(* PLC project One Station VGP, Blank VGP 1.0 *)
(* stored: creationDateTime 2016-05-18T21:14:07, modificationDateTime 2020-03-26T18:29:31 *)

FUNCTION ConvertPressure : SINT
  VAR_INPUT
    Pressure_input : UINT;
  END_VAR
  VAR_OUTPUT
    Pressure_output : INT;
  END_VAR
  VAR
    Pressure_real : LREAL;
  END_VAR

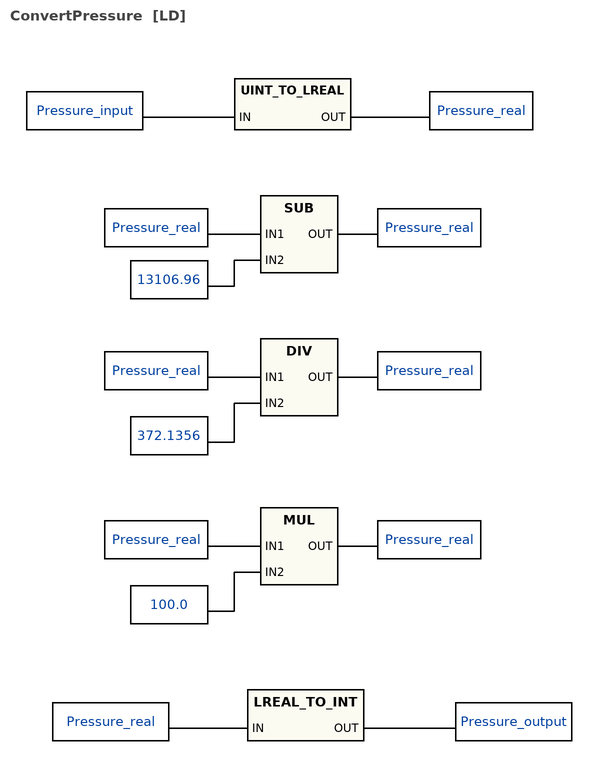
(* LD diagram, written out as Structured Text *)
Pressure_real := UINT_TO_LREAL(Pressure_input);
Pressure_real := Pressure_real - 13106.96;
Pressure_real := Pressure_real / 372.1356;
Pressure_real := Pressure_real * 100.0;
Pressure_output := LREAL_TO_INT(Pressure_real);
END_FUNCTION

PROGRAM My_Program
  VAR
    pressure AT %IW0 : UINT;
    pressure_psi AT %QW6 : INT;
    min_sp AT %QW1 : INT;
    max_sp AT %QW2 : INT;
  END_VAR
  VAR
    pump_mode : BOOL;
    pm_pump : BOOL;
    pm_valve : BOOL;
    valve_mode : BOOL;
    vm_pump : BOOL;
    vm_valve : BOOL;
    manual_mode : BOOL;
    mm_pump : BOOL;
    mm_valve : BOOL;
  END_VAR
  VAR
    mode_register AT %QW3 : INT;
    pump_register AT %QW4 : INT;
    valve_register AT %QW5 : INT;
  END_VAR
  VAR
    over_pressure : BOOL;
  END_VAR
  VAR
    pump AT %QX0.0 : BOOL;
    valve AT %QX0.1 : BOOL;
  END_VAR
  VAR
    TOF0 : TOF;
  END_VAR
  VAR  (* added by the conversion: wires and edge detectors of the diagram *)
    _LE4_ENO : BOOL;
    _LE4_OUT : BOOL;
    _GE11_ENO : BOOL;
    _GE11_OUT : BOOL;
    _LE22_ENO : BOOL;
    _LE22_OUT : BOOL;
    _GE29_ENO : BOOL;
    _GE29_OUT : BOOL;
    _EQ44_ENO : BOOL;
    _EQ44_OUT : BOOL;
    _EQ50_ENO : BOOL;
    _EQ50_OUT : BOOL;
    _ConvertPressure99_Pressure_output : ANY;
    _ConvertPressure99_OUT : SINT;
  END_VAR

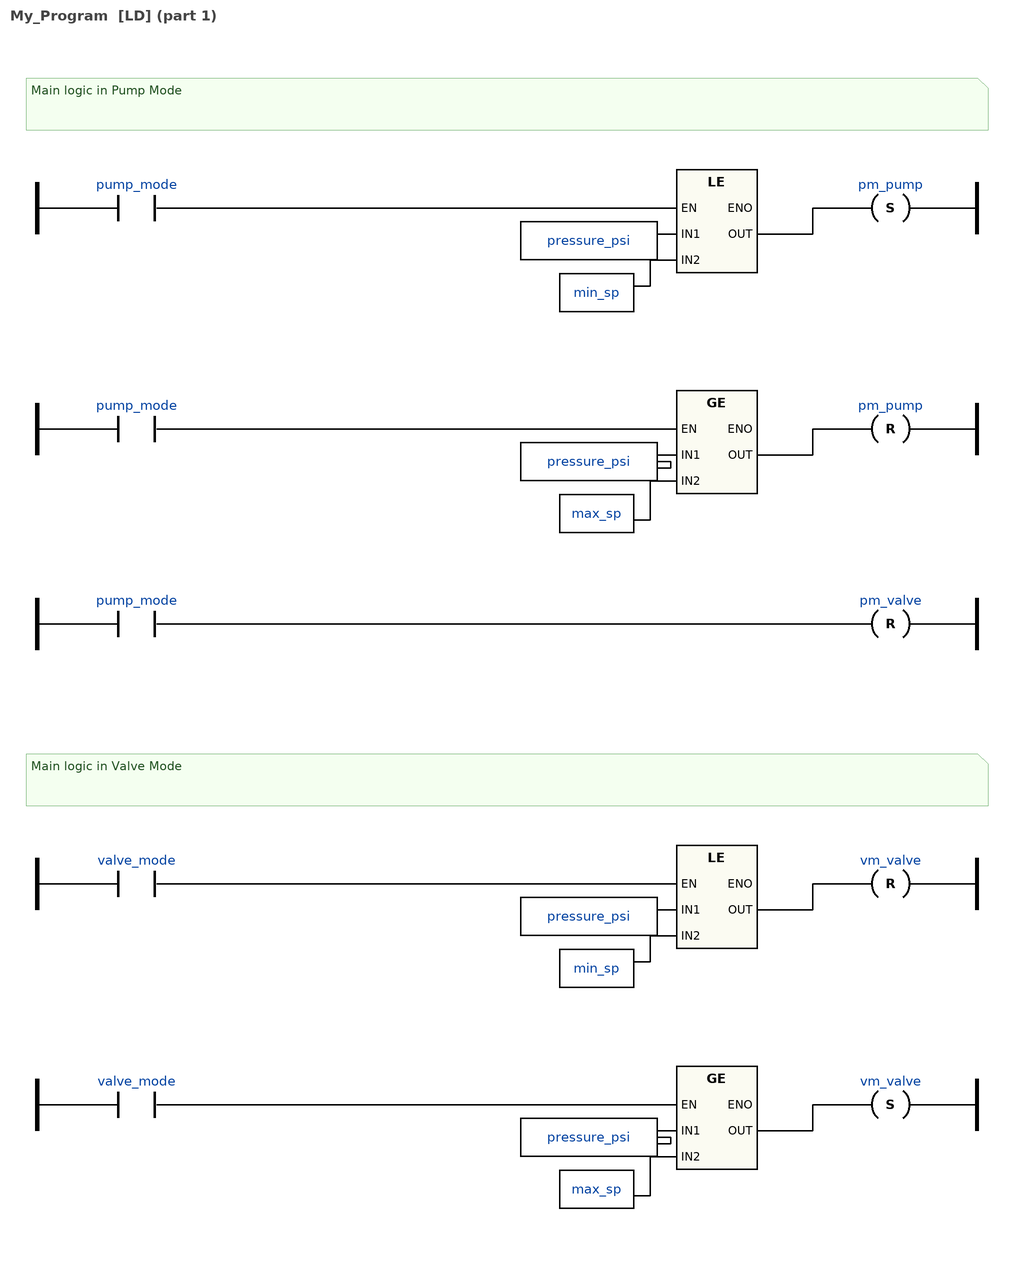
(* LD diagram, written out as Structured Text *)
(* Main logic in Pump Mode *)
_LE4_OUT := LE(EN := pump_mode, IN1 := pressure_psi, IN2 := min_sp, ENO => _LE4_ENO);
IF _LE4_OUT THEN pm_pump := TRUE; END_IF;
_GE11_OUT := GE(EN := pump_mode, IN1 := pressure_psi, IN2 := max_sp, ENO => _GE11_ENO);
IF _GE11_OUT THEN pm_pump := FALSE; END_IF;
IF pump_mode THEN pm_valve := FALSE; END_IF;
(* Main logic in Valve Mode *)
_LE22_OUT := LE(EN := valve_mode, IN1 := pressure_psi, IN2 := min_sp, ENO => _LE22_ENO);
IF _LE22_OUT THEN vm_valve := FALSE; END_IF;
_GE29_OUT := GE(EN := valve_mode, IN1 := pressure_psi, IN2 := max_sp, ENO => _GE29_ENO);
IF _GE29_OUT THEN vm_valve := TRUE; END_IF;
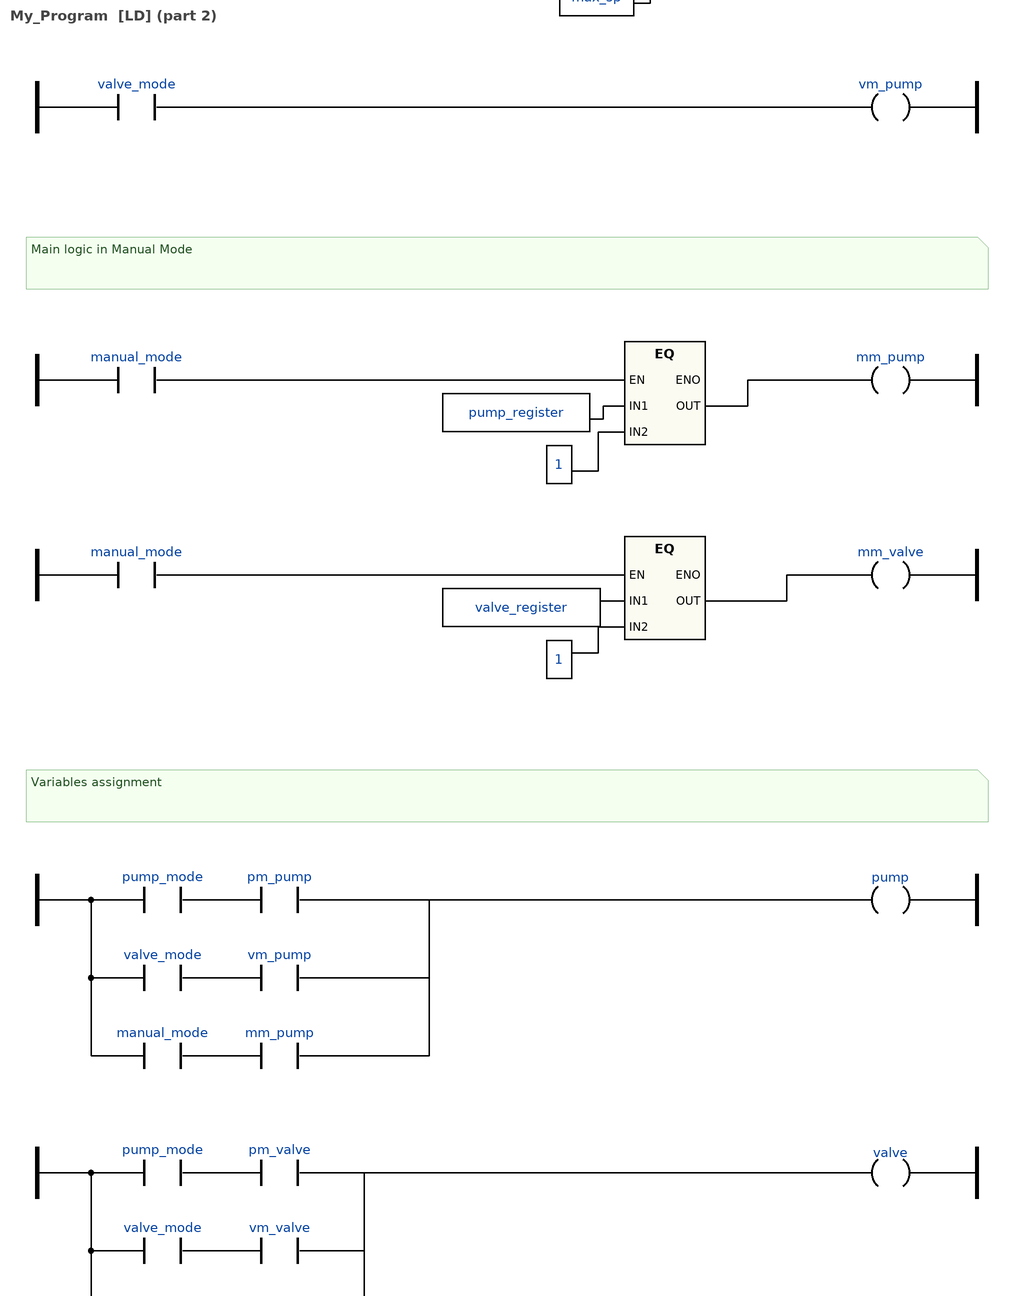
vm_pump := valve_mode;
(* Main logic in Manual Mode *)
_EQ44_OUT := EQ(EN := manual_mode, IN1 := pump_register, IN2 := 1, ENO => _EQ44_ENO);
mm_pump := _EQ44_OUT;
_EQ50_OUT := EQ(EN := manual_mode, IN1 := valve_register, IN2 := 1, ENO => _EQ50_ENO);
mm_valve := _EQ50_OUT;
(* Variables assignment *)
pump := pump_mode AND pm_pump OR valve_mode AND vm_pump OR manual_mode AND mm_pump;
valve := pump_mode AND pm_valve OR valve_mode AND vm_valve OR manual_mode AND mm_valve;
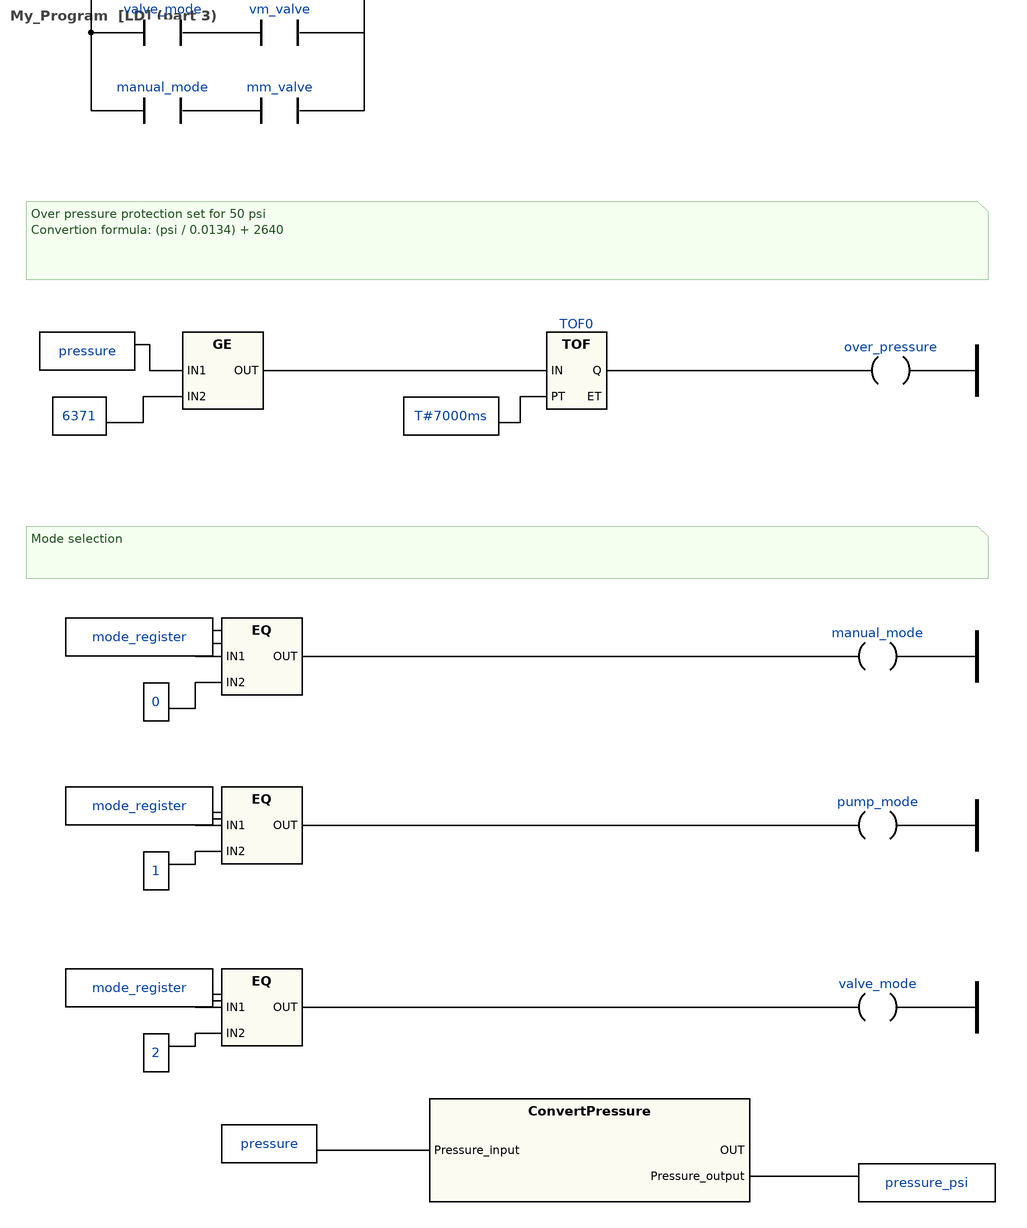
(* Over pressure protection set for 50 psi
Convertion formula: (psi / 0.0134) + 2640 *)
TOF0(IN := pressure >= 6371, PT := T#7000ms);
over_pressure := TOF0.Q;
(* Mode selection *)
manual_mode := mode_register = 0;
pump_mode := mode_register = 1;
valve_mode := mode_register = 2;
_ConvertPressure99_OUT := ConvertPressure(Pressure_input := pressure, Pressure_output => _ConvertPressure99_Pressure_output);
pressure_psi := _ConvertPressure99_Pressure_output;
END_PROGRAM

CONFIGURATION Config0
  RESOURCE Res0 ON PLC
    TASK TaskMain(INTERVAL := T#50ms, PRIORITY := 0);
    PROGRAM Inst0 WITH TaskMain : My_Program;
  END_RESOURCE
END_CONFIGURATION
